// TIA Portal V17 export
// export: Created 2023-02-13T11:16:25.2508372Z, ExportSetting WithDefaults, DisplayName Totally Integrated Automation Portal, DisplayVersion V17, DisplayName TIA Portal Openness, DisplayVersion V17, DisplayName TIA Portal Teamcenter Gateway, DisplayVersion V17, DisplayName TIA Portal Version Control Interface, DisplayVersion V17, DisplayName SINAMICS Startdrive Advanced, DisplayVersion V17, DisplayName SINAMICS Startdrive G130, G150, S120, S150, SINAMICS MV, S210, DisplayVersion V17, DisplayName SINAMICS Startdrive G110M, G120, G120C, G120D, G120P, G115D, DisplayVersion V17, DisplayName STEP 7 Professional, DisplayVersion V17, DisplayName STEP 7 Safety, DisplayVersion V17, DisplayName WinCC Professional, DisplayVersion V17
FUNCTION_BLOCK "IO_Digital_Storage"   // FB22, LAD
{ S7_Optimized_Access := 'TRUE' }
VERSION : 0.1
// stored: AutoNumber false, IsIECCheckEnabled false, IsRetainMemResEnabled false, MemoryReserve 100, SetENOAutomatically false, UDAEnableTagReadback false
   VAR_INPUT
      lock : Bool;
      init : Bool;
      Reset : Bool;
   END_VAR
   VAR
      "FS-23.01" : "Digital";
      "FS-24.01" { S7_SetPoint := 'True'} : "Digital";
      "FS-34.01" { S7_SetPoint := 'True'} : "Digital";
      "FS-35.01" { S7_SetPoint := 'True'} : "Digital";
   END_VAR
BEGIN

REGION Network 1: FS-23.01
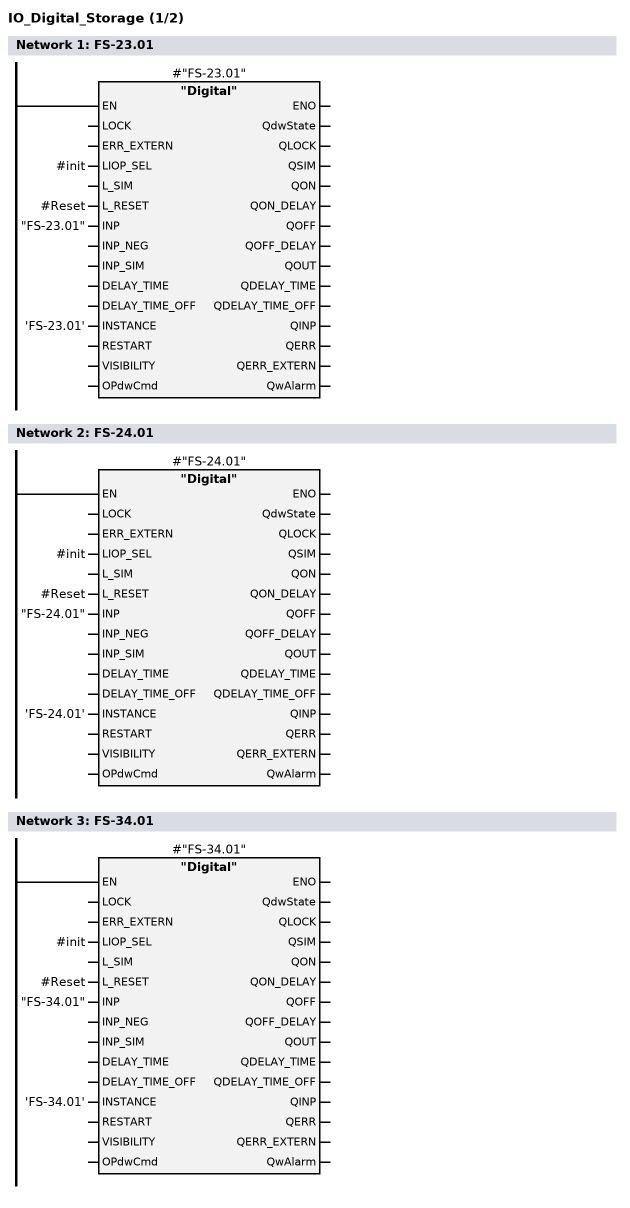
   RUNG wire#powerrail
      #"FS-23.01"(LOCK :=, ERR_EXTERN :=, LIOP_SEL := #init, L_SIM :=, L_RESET := #Reset, INP := "FS-23.01", INP_NEG :=, INP_SIM :=, DELAY_TIME :=, DELAY_TIME_OFF :=, INSTANCE := 'FS-23.01', RESTART :=, VISIBILITY :=, OPdwCmd :=, QdwState =>, QLOCK =>, QSIM =>, QON =>, QON_DELAY =>, QOFF =>, QOFF_DELAY =>, QOUT =>, QDELAY_TIME =>, QDELAY_TIME_OFF =>, QINP =>, QERR =>, QERR_EXTERN =>, QwAlarm =>)
   END_RUNG
   // the same network as SCL:
   #"FS-23.01"(LIOP_SEL := #init, L_RESET := #Reset, INP := "FS-23.01", INSTANCE := 'FS-23.01');   // "Digital"
END_REGION

REGION Network 2: FS-24.01
   RUNG wire#powerrail
      #"FS-24.01"(LOCK :=, ERR_EXTERN :=, LIOP_SEL := #init, L_SIM :=, L_RESET := #Reset, INP := "FS-24.01", INP_NEG :=, INP_SIM :=, DELAY_TIME :=, DELAY_TIME_OFF :=, INSTANCE := 'FS-24.01', RESTART :=, VISIBILITY :=, OPdwCmd :=, QdwState =>, QLOCK =>, QSIM =>, QON =>, QON_DELAY =>, QOFF =>, QOFF_DELAY =>, QOUT =>, QDELAY_TIME =>, QDELAY_TIME_OFF =>, QINP =>, QERR =>, QERR_EXTERN =>, QwAlarm =>)
   END_RUNG
   // the same network as SCL:
   #"FS-24.01"(LIOP_SEL := #init, L_RESET := #Reset, INP := "FS-24.01", INSTANCE := 'FS-24.01');   // "Digital"
END_REGION

REGION Network 3: FS-34.01
   RUNG wire#powerrail
      #"FS-34.01"(LOCK :=, ERR_EXTERN :=, LIOP_SEL := #init, L_SIM :=, L_RESET := #Reset, INP := "FS-34.01", INP_NEG :=, INP_SIM :=, DELAY_TIME :=, DELAY_TIME_OFF :=, INSTANCE := 'FS-34.01', RESTART :=, VISIBILITY :=, OPdwCmd :=, QdwState =>, QLOCK =>, QSIM =>, QON =>, QON_DELAY =>, QOFF =>, QOFF_DELAY =>, QOUT =>, QDELAY_TIME =>, QDELAY_TIME_OFF =>, QINP =>, QERR =>, QERR_EXTERN =>, QwAlarm =>)
   END_RUNG
   // the same network as SCL:
   #"FS-34.01"(LIOP_SEL := #init, L_RESET := #Reset, INP := "FS-34.01", INSTANCE := 'FS-34.01');   // "Digital"
END_REGION

REGION Network 4: FS-35.01
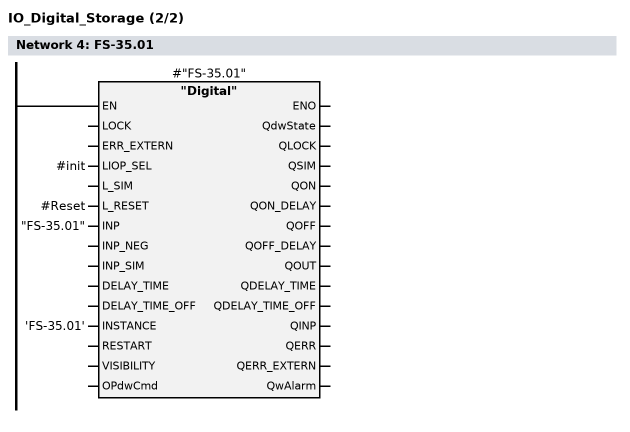
   RUNG wire#powerrail
      #"FS-35.01"(LOCK :=, ERR_EXTERN :=, LIOP_SEL := #init, L_SIM :=, L_RESET := #Reset, INP := "FS-35.01", INP_NEG :=, INP_SIM :=, DELAY_TIME :=, DELAY_TIME_OFF :=, INSTANCE := 'FS-35.01', RESTART :=, VISIBILITY :=, OPdwCmd :=, QdwState =>, QLOCK =>, QSIM =>, QON =>, QON_DELAY =>, QOFF =>, QOFF_DELAY =>, QOUT =>, QDELAY_TIME =>, QDELAY_TIME_OFF =>, QINP =>, QERR =>, QERR_EXTERN =>, QwAlarm =>)
   END_RUNG
   // the same network as SCL:
   #"FS-35.01"(LIOP_SEL := #init, L_RESET := #Reset, INP := "FS-35.01", INSTANCE := 'FS-35.01');   // "Digital"
END_REGION
END_FUNCTION_BLOCK
